FUNCTION TryConvert_DINT_TO_UINT : BOOL
VAR_INPUT
	in : DINT;
	out : REFERENCE TO UINT;
END_VAR

IF in > DatatypeLimits.MAX_VALUE_OF_DINT_WHICH_CAN_BE_HELD_IN_A_UINT THEN
	RETURN;
END_IF

IF in < DatatypeLimits.MIN_VALUE_OF_DINT_WHICH_CAN_BE_HELD_IN_A_UINT THEN
	RETURN;
END_IF

out := DINT_TO_UINT(in);
TryConvert_DINT_TO_UINT := TRUE;

END_FUNCTION

(* stored: Version 1.1.0.1, ProductVersion 3.1.4024.12
   POU TryConvert_DINT_TO_UINT: Id {da922240-5dcf-4a08-ae85-ad34046485f2}, SpecialFunc None *)
